// TwinCAT 3 PLC project Untitled1
// ProgramVersion: 3.1.4024.0
// libraries:
//   Tc2_Standard, * (Beckhoff Automation GmbH)
//   Tc2_System, * (Beckhoff Automation GmbH)
//   Tc3_Module, * (Beckhoff Automation GmbH)
//   VisuSymbols,3.5.10.0,System
// project tree:
//   / GlobalTextList.TcGTLO, PlcTask.TcTTO, PlcTask2.TcTTO, Visualization Manager.TcVMO (not stored)
//   GVLs/ GVL.TcGVL
//   POUs/ MAIN.TcPOU, POU.TcPOU, CaseStruct.TcPOU
//   VISUs/ Visualization.TcVIS
// real-time tasks:
//   TASK PlcTask: cycle T#2000ms, priority 20, ADS port 350
//   TASK PlcTask2: cycle T#5ms, priority 19, ADS port 351

CONFIGURATION Untitled1
    RESOURCE PLC ON TwinCAT3
        TASK PlcTask(INTERVAL := T#10ms, PRIORITY := 20);
        TASK PlcTask2(INTERVAL := T#5ms, PRIORITY := 19);
        PROGRAM MAIN WITH PlcTask : MAIN;
        PROGRAM CaseStruct WITH PlcTask2 : CaseStruct;
    END_RESOURCE
END_CONFIGURATION

// ---- GVLs/GVL.TcGVL
{attribute 'qualified_only'}
VAR_GLOBAL
	// Case structure
	caseInput : INT := 0;
	
	// Variabelen
	ProductGedetecteerd1 : BOOL;	
	ProductGedetecteerd2 : BOOL;
	MotorStatus : BOOL;

	// Timers
	Timer : TON;
	TimerOn : BOOL := FALSE;
END_VAR

// ---- POUs/MAIN.TcPOU
PROGRAM MAIN
VAR
	Afstand: INT;
	TransportBandSnelheid : REAL;
	KlaarVoorVolgende : BOOL;
	// Timers
	Timer : TON;
	TimerOn : BOOL := FALSE;
END_VAR

Timer(IN := TimerOn, PT := T#30S); // Start de timer voor 30 seconden

// Case 1: Productdetectie (detecteer producten op de band en start de motor).
IF GVL.caseInput = 1 THEN // Controleer of het eerste product gedetecteerd is en het tweede niet
    GVL.MotorStatus := TRUE; // Zet de motorstatus aan (start de motor)
END_IF

// Case 2: Als de motor aan staat moet een timer gaan lopen die de tijd opneemt hoe lang de band loopt.
IF GVL.caseInput = 2 THEN
	TimerOn := TRUE; // Start de timer.
	IF Timer.ET > T#1S THEN // Controleer of de band langer als een seconde loopt
		GVL.ProductGedetecteerd1 := FALSE; // Zet de sensor productgedetecteerd uit
	END_IF
END_IF

// Case 3: Stoppen van de band (stop de motor na het bereiken van het einddoel).
IF GVL.caseInput = 3 THEN // Controleer of het tweede product gedetecteerd is en de band al langer als een seconde loopt
    IF GVL.MotorStatus THEN
		POU(Timer.ET, Afstand); // Geef de afstand en tijd wat het object er over heeft gedaan mee aan de functie
	END_IF 
	GVL.MotorStatus := 0; // Zet de motorstatus uit (stop de motor)
	TimerOn := FALSE;
	KlaarVoorVolgende := TRUE;
END_IF

END_PROGRAM

// ---- POUs/POU.TcPOU
FUNCTION POU : BOOL
VAR_INPUT
 Tijd : TIME;
 Afstand : INT;
END_VAR
VAR
	TijdInSeconden : REAL;
	TransportbandSnelheid : REAL;
END_VAR

TijdInSeconden := TIME_TO_REAL(Tijd)/1000; // Zet de tijd om naar een REAL waarde in seconden

IF Afstand = 0 THEN // Controleer of de afstand gelijk is aan 0
    TransportBandSnelheid := 0; // Stel de transportbandsnelheid in op 0
ELSE	
    TransportBandSnelheid := Afstand / TijdInSeconden; // Bereken de snelheid van het transportband
END_IF

END_FUNCTION

// ---- POUs/CaseStruct.TcPOU
PROGRAM CaseStruct
VAR

END_VAR

CASE GVL.caseInput OF 
	0: // Initialisatie.
		GVL.ProductGedetecteerd1 := FALSE;	
		GVL.ProductGedetecteerd2 := FALSE;
		GVL.MotorStatus := FALSE;
		IF GVL.ProductGedetecteerd1 AND NOT GVL.ProductGedetecteerd2 THEN
			GVL.caseInput := 1;
		END_IF
	1: // Product aan de start gedetecteerd.
		IF GVL.MotorStatus THEN
			GVL.caseInput := 2;
		END_IF
	2: // Product op het einde gedetecteerd.
		IF GVL.ProductGedetecteerd2 AND MAIN.Timer.ET > T#1S THEN
			GVL.caseInput := 3;
		END_IF
	3: // Programma weer afsluiten.
		IF MAIN.KlaarVoorVolgende THEN
			GVL.caseInput := 1;
			MAIN.KlaarVoorVolgende := FALSE;
		END_IF
END_CASE

END_PROGRAM

// ---- GlobalTextList.TcGTLO
TEXTLIST GlobalTextList
  103 = '0m                  Afstand                         100m'
  560 = '0m          Afstand            100m'
  623 = '0m          Afstand     100m'
  478 = '0m  Afstand     100m'
  286 = '0m  Afstand  100m'
  101 = 'Afstand'
  786 = 'Motor status'
  268 = 'Sensor 1'
  529 = 'Sensor 1\n(Begin band)'
  554 = 'Sensor 2'
  400 = 'Sensor 2\n(Einde band)'
  322 = 'Transportband snelheid m/s'
END_TEXTLIST

// ---- VISUs/Visualization.TcVIS
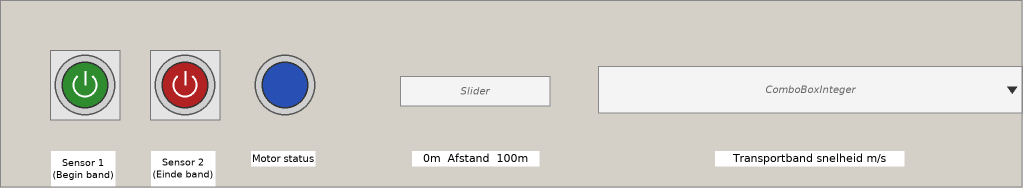
VISUALIZATION Visualization  // 1023x188
    Lamp1 (250,50 70x70), variable: GVL.MotorStatus, style: Lamp-Lamp1-Blue
    PowerSwitch (50,50 70x70), variable: GVL.ProductGedetecteerd1, behaviour: TOGGLE, style: Switch-PowerSwitch-Green
    PowerSwitch (150,50 70x70), variable: GVL.ProductGedetecteerd2, behaviour: TOGGLE, style: Switch-PowerSwitch-Red
    Slider (400,76 150x30), variable: StopBeld.Afstand, scale 0..100
    Textfield (50,150 66x38), "Sensor 1 (Begin band)"
    Textfield (150,150 66x37), "Sensor 2 (Einde band)"
    Textfield (250,150 66x17), "Motor status"
    Textfield (411,150 129x17), "0m Afstand 100m"
    ComboBoxInteger (598,66 425x47), variable: GVL.TransportBandSnelheid, text list: GVL.TransportBandSnelheid
    Textfield (714,150 191x17), "Transportband snelheid m/s"
END_VISUALIZATION
